Yaskawa INFORM job: Print3D.JBI

/JOB
//NAME Print3D
//POS
///NPOS 538,0,0,0,0,0
///TOOL 9
///POSTYPE PULSE
///PULSE
C00000=-32438,37072,-110539,-86183,-121616,78041,0
C00001=-32438,56188,-108455,-81750,-115935,87656,0
C00002=-32438,56821,-108216,-81665,-115782,87885,0
C00003=-32406,57586,-105976,-81950,-116211,87210,0
C00004=-32348,57787,-105393,-82074,-116292,87030,0
C00005=-31898,58636,-102954,-82798,-116500,86260,0
C00006=-31753,58820,-102432,-83000,-116512,86091,0
C00007=-30966,59540,-100399,-83997,-116406,85414,0
C00008=-30755,59682,-100001,-84246,-116346,85275,0
C00009=-29730,60178,-98619,-85379,-115942,84773,0
C00010=-29476,60259,-98393,-85644,-115819,84683,0
C00011=-28322,60462,-97831,-86792,-115175,84417,0
C00012=-28051,60472,-97803,-87049,-115007,84386,0
C00013=-26882,60354,-98131,-88113,-114216,84389,0
C00014=-26621,60290,-98306,-88341,-114026,84422,0
C00015=-25550,59868,-99482,-89239,-113195,84693,0
C00016=-25325,59740,-99839,-89419,-113009,84784,0
C00017=-24465,59071,-101720,-90078,-112243,85290,0
C00018=-24300,58897,-102214,-90195,-112083,85429,0
C00019=-20558,65330,-84764,-76831,-126138,82193,0
C00020=-20473,65073,-85436,-76785,-125928,82368,0
C00021=-20281,63933,-88440,-76413,-125114,83185,0
C00022=-20280,63674,-89129,-76290,-124955,83380,0
C00023=-20473,62589,-92031,-75590,-124397,84229,0
C00024=-20562,62357,-92656,-75394,-124304,84420,0
C00025=-20633,62241,-92968,-75270,-124274,84519,0
C00026=-21140,61448,-95121,-74399,-124058,85205,0
C00027=-21314,61269,-95612,-74142,-124041,85371,0
C00028=-22223,60633,-97359,-72935,-124133,86005,0
C00029=-22461,60524,-97659,-72644,-124194,86127,0
C00030=-23585,60225,-98488,-71363,-124621,86540,0
C00031=-23855,60198,-98563,-71076,-124755,86605,0
C00032=-25034,60265,-98378,-69905,-125482,86749,0
C00033=-25297,60322,-98219,-69665,-125679,86750,0
C00034=-30759,54831,-114236,-82744,-113724,89580,0
C00035=-30996,54948,-113875,-82536,-113911,89487,0
C00036=-31840,55566,-111976,-81865,-114711,88973,0
C00037=-31986,55730,-111478,-81769,-114886,88834,0
C00038=-32400,56520,-109107,-81604,-115582,88151,0
C00039=-32443,56714,-108532,-81625,-115721,87982,0
C00040=-32441,56759,-108398,-81642,-115746,87941,0
C00041=-26549,59218,-101304,-88131,-113571,85310,0
C00042=-26104,59051,-101778,-88513,-113235,85419,0
C00043=-25336,58461,-103455,-89105,-112549,85871,0
C00044=-24860,57729,-105559,-89395,-111996,86479,0
C00045=-21345,63810,-88769,-75336,-125745,83446,0
C00046=-21533,62838,-91363,-74678,-125240,84207,0
C00047=-22059,62019,-93570,-73765,-125019,84912,0
C00048=-22866,61443,-95135,-72683,-125107,85482,0
C00049=-23853,61172,-95878,-71559,-125500,85853,0
C00050=-24885,61232,-95712,-70546,-126159,85983,0
C00051=-30057,55478,-112245,-83650,-113759,88907,0
C00052=-30815,56036,-110556,-83049,-114467,88450,0
C00053=-31204,56744,-108442,-82877,-115075,87841,0
C00054=-31195,57522,-106160,-83130,-115500,87151,0
C00055=-30810,58276,-103983,-83747,-115680,86464,0
C00056=-30111,58912,-102170,-84625,-115587,85860,0
C00057=-29186,59348,-100939,-85647,-115233,85412,0
C00058=-28137,59526,-100438,-86701,-114669,85174,0
C00059=-27073,59422,-100730,-87686,-113973,85177,0
C00060=-26627,59248,-101220,-88065,-113630,85290,0
C00061=-26503,59292,-101097,-88193,-113572,85244,0
C00062=-26043,59118,-101588,-88588,-113223,85358,0
C00063=-25248,58507,-103322,-89200,-112515,85825,0
C00064=-24755,57750,-105498,-89502,-111944,86454,0
C00065=-21248,63808,-88772,-75428,-125681,83432,0
C00066=-21442,62804,-91454,-74751,-125159,84218,0
C00067=-21984,61958,-93735,-73809,-124930,84946,0
C00068=-22819,61364,-95353,-72691,-125021,85536,0
C00069=-23841,61083,-96120,-71527,-125427,85919,0
C00070=-24910,61146,-95949,-70477,-126107,86053,0
C00071=-30130,55424,-112411,-83560,-113765,88964,0
C00072=-30914,56000,-110664,-82939,-114497,88492,0
C00073=-31314,56732,-108479,-82763,-115127,87862,0
C00074=-31302,57536,-106119,-83029,-115568,87149,0
C00075=-30903,58316,-103868,-83669,-115753,86438,0
C00076=-30180,58974,-101994,-84577,-115657,85813,0
C00077=-29224,59426,-100721,-85633,-115291,85350,0
C00078=-28141,59610,-100203,-86721,-114708,85105,0
C00079=-27043,59502,-100505,-87735,-113986,85108,0
C00080=-26582,59322,-101013,-88127,-113631,85225,0
C00081=-26458,59365,-100890,-88255,-113573,85179,0
C00082=-25982,59185,-101398,-88663,-113212,85297,0
C00083=-25161,58554,-103189,-89294,-112480,85779,0
C00084=-21320,64890,-85917,-75895,-126401,82640,0
C00085=-21152,63807,-88776,-75520,-125616,83417,0
C00086=-21351,62770,-91544,-74823,-125078,84229,0
C00087=-21910,61897,-93900,-73853,-124843,84981,0
C00088=-22772,61284,-95570,-72699,-124936,85589,0
C00089=-23829,60995,-96362,-71495,-125353,85984,0
C00090=-24935,61060,-96185,-70408,-126055,86123,0
C00091=-30204,55370,-112576,-83469,-113771,89021,0
C00092=-31012,55964,-110771,-82828,-114527,88533,0
C00093=-31424,56720,-108515,-82649,-115180,87883,0
C00094=-31410,57551,-106078,-82927,-115635,87146,0
C00095=-30995,58356,-103753,-83591,-115828,86412,0
C00096=-30249,59037,-101817,-84530,-115728,85767,0
C00097=-29263,59503,-100502,-85620,-115350,85289,0
C00098=-28146,59694,-99968,-86740,-114746,85036,0
C00099=-27014,59583,-100279,-87785,-114000,85038,0
C00100=-26536,59395,-100806,-88189,-113632,85159,0
C00101=-26414,59439,-100683,-88316,-113573,85114,0
C00102=-25921,59252,-101208,-88737,-113200,85235,0
C00103=-25074,58601,-103056,-89388,-112445,85733,0
C00104=-21231,64924,-85829,-75997,-126360,82601,0
C00105=-21056,63806,-88778,-75612,-125552,83403,0
C00106=-21259,62736,-91634,-74896,-124997,84240,0
C00107=-21835,61837,-94064,-73898,-124755,85015,0
C00108=-22725,61205,-95786,-72707,-124850,85642,0
C00109=-23817,60907,-96603,-71464,-125280,86050,0
C00110=-24961,60974,-96420,-70339,-126003,86193,0
C00111=-30277,55316,-112741,-83379,-113776,89078,0
C00112=-31111,55928,-110879,-82718,-114558,88574,0
C00113=-31534,56708,-108550,-82535,-115232,87903,0
C00114=-31517,57565,-106036,-82825,-115703,87144,0
C00115=-31088,58397,-103638,-83513,-115903,86386,0
C00116=-30317,59099,-101640,-84484,-115799,85720,0
C00117=-29301,59581,-100284,-85607,-115409,85227,0
C00118=-28150,59778,-99732,-86759,-114784,84966,0
C00119=-26984,59663,-100054,-87834,-114014,84969,0
C00120=-26491,59469,-100598,-88250,-113633,85094,0
C00121=-26332,59013,-101884,-88286,-113359,85467,0
C00122=-24985,57748,-105506,-89278,-112076,86471,0
C00123=-24944,57669,-105734,-89300,-112022,86537,0
C00124=-21511,64356,-87324,-75447,-126200,83067,0
C00125=-25467,58473,-103419,-88982,-112632,85869,0
C00126=-25645,58607,-103036,-88843,-112789,85766,0
C00127=-21453,63977,-88326,-75315,-125923,83339,0
C00128=-21420,63763,-88894,-75241,-125765,83493,0
C00129=-21433,63691,-89084,-75193,-125729,83550,0
C00130=-25822,58743,-102651,-88706,-112947,85662,0
C00131=-25998,58879,-102263,-88572,-113105,85557,0
C00132=-21465,63524,-89527,-75080,-125643,83679,0
C00133=-21497,63359,-89968,-74968,-125557,83808,0
C00134=-26173,59017,-101873,-88439,-113264,85453,0
C00135=-26184,59026,-101848,-88430,-113274,85446,0
C00136=-26310,59073,-101715,-88322,-113368,85415,0
C00137=-21529,63194,-90407,-74856,-125472,83937,0
C00138=-21562,63031,-90844,-74745,-125386,84066,0
C00139=-26443,59123,-101573,-88207,-113470,85382,0
C00140=-26577,59174,-101429,-88093,-113571,85349,0
C00141=-21595,62868,-91280,-74634,-125299,84193,0
C00142=-21603,62825,-91397,-74604,-125276,84227,0
C00143=-21648,62753,-91590,-74525,-125258,84289,0
C00144=-26710,59225,-101285,-87979,-113672,85316,0
C00145=-26843,59277,-101140,-87866,-113774,85282,0
C00146=-21710,62654,-91854,-74417,-125232,84374,0
C00147=-21772,62557,-92118,-74308,-125205,84457,0
C00148=-26976,59328,-100994,-87753,-113876,85249,0
C00149=-27108,59381,-100847,-87641,-113978,85215,0
C00150=-21835,62459,-92380,-74200,-125179,84541,0
C00151=-21897,62362,-92642,-74091,-125153,84625,0
C00152=-27224,59395,-100808,-87534,-114055,85212,0
C00153=-27339,59405,-100778,-87428,-114129,85212,0
C00154=-21960,62265,-92903,-73983,-125127,84708,0
C00155=-22023,62169,-93163,-73874,-125101,84791,0
C00156=-27453,59416,-100747,-87322,-114204,85212,0
C00157=-27568,59427,-100716,-87216,-114278,85212,0
C00158=-22086,62073,-93422,-73765,-125074,84875,0
C00159=-22112,62034,-93528,-73720,-125063,84909,0
C00160=-22159,61999,-93623,-73656,-125068,84943,0
C00161=-27682,59438,-100685,-87110,-114353,85212,0
C00162=-27796,59450,-100653,-87005,-114428,85211,0
C00163=-22240,61941,-93782,-73548,-125078,85001,0
C00164=-22321,61882,-93941,-73440,-125087,85058,0
C00165=-27910,59461,-100621,-86899,-114503,85210,0
C00166=-28024,59473,-100588,-86794,-114578,85210,0
C00167=-22402,61824,-94100,-73331,-125095,85116,0
C00168=-22483,61766,-94257,-73222,-125104,85173,0
C00169=-28138,59485,-100555,-86688,-114653,85209,0
C00170=-28149,59486,-100552,-86678,-114660,85209,0
C00171=-28242,59469,-100598,-86585,-114710,85231,0
C00172=-22564,61708,-94415,-73113,-125113,85231,0
C00173=-22645,61650,-94572,-73004,-125122,85288,0
C00174=-28344,59452,-100648,-86483,-114765,85254,0
C00175=-28446,59434,-100698,-86380,-114820,85277,0
C00176=-22727,61592,-94728,-72895,-125130,85346,0
C00177=-22809,61535,-94884,-72785,-125140,85402,0
C00178=-28549,59416,-100747,-86277,-114875,85300,0
C00179=-28651,59399,-100796,-86174,-114929,85324,0
C00180=-22891,61478,-95039,-72675,-125149,85459,0
C00181=-22987,61451,-95114,-72566,-125187,85496,0
C00182=-28754,59382,-100845,-86071,-114985,85347,0
C00183=-28856,59364,-100893,-85968,-115040,85370,0
C00184=-23082,61424,-95188,-72457,-125225,85532,0
C00185=-23179,61397,-95262,-72348,-125263,85569,0
C00186=-28959,59347,-100941,-85865,-115095,85393,0
C00187=-29062,59331,-100988,-85761,-115150,85416,0
C00188=-23275,61370,-95335,-72238,-125302,85606,0
C00189=-23371,61343,-95408,-72129,-125340,85642,0
C00190=-29164,59314,-101036,-85658,-115204,85438,0
C00191=-29257,59269,-101162,-85556,-115240,85484,0
C00192=-23467,61317,-95480,-72019,-125379,85678,0
C00193=-23564,61291,-95552,-71909,-125417,85714,0
C00194=-29349,59224,-101287,-85454,-115276,85530,0
C00195=-29442,59180,-101412,-85351,-115312,85575,0
C00196=-23660,61264,-95623,-71799,-125454,85750,0
C00197=-23757,61239,-95694,-71689,-125494,85786,0
C00198=-29535,59136,-101537,-85249,-115348,85620,0
C00199=-29628,59092,-101661,-85146,-115383,85665,0
C00200=-23855,61216,-95757,-71579,-125535,85820,0
C00201=-23966,61222,-95741,-71470,-125605,85834,0
C00202=-29721,59048,-101784,-85043,-115418,85710,0
C00203=-29815,59005,-101908,-84939,-115453,85755,0
C00204=-24076,61228,-95725,-71362,-125675,85848,0
C00205=-24187,61234,-95708,-71253,-125746,85862,0
C00206=-29908,58961,-102031,-84836,-115489,85800,0
C00207=-30002,58918,-102153,-84732,-115525,85845,0
C00208=-24298,61240,-95691,-71144,-125816,85876,0
C00209=-24409,61246,-95673,-71036,-125888,85890,0
C00210=-30091,58861,-102314,-84628,-115550,85901,0
C00211=-30173,58785,-102531,-84525,-115561,85973,0
C00212=-24519,61253,-95655,-70927,-125959,85904,0
C00213=-24630,61260,-95636,-70819,-126029,85918,0
C00214=-30256,58709,-102748,-84422,-115573,86045,0
C00215=-30338,58633,-102964,-84318,-115584,86117,0
C00216=-24741,61267,-95617,-70711,-126100,85931,0
C00217=-24841,61273,-95599,-70612,-126165,85944,0
C00218=-24853,61278,-95586,-70603,-126176,85942,0
C00219=-30421,58557,-103180,-84214,-115595,86188,0
C00220=-30504,58482,-103395,-84110,-115606,86260,0
C00221=-24982,61330,-95443,-70498,-126292,85925,0
C00222=-29264,55260,-112912,-84393,-113237,89051,0
C00223=-30587,58407,-103609,-84006,-115617,86331,0
C00224=-30671,58332,-103822,-83900,-115628,86403,0
C00225=-29407,55307,-112767,-84261,-113335,89018,0
C00226=-29550,55355,-112622,-84129,-113433,88983,0
C00227=-30749,58243,-104079,-83796,-115628,86487,0
C00228=-30814,58113,-104451,-83692,-115598,86604,0
C00229=-29693,55402,-112476,-83998,-113532,88949,0
C00230=-29835,55450,-112329,-83868,-113631,88915,0
C00231=-30878,57985,-104821,-83589,-115567,86721,0
C00232=-30943,57857,-105191,-83485,-115537,86837,0
C00233=-29979,55504,-112166,-83737,-113734,88876,0
C00234=-30155,55630,-111781,-83595,-113896,88772,0
C00235=-31008,57729,-105559,-83380,-115507,86954,0
C00236=-31074,57603,-105926,-83275,-115476,87070,0
C00237=-30331,55758,-111394,-83455,-114058,88667,0
C00238=-30505,55887,-111005,-83317,-114221,88561,0
C00239=-31104,57379,-106577,-83175,-115372,87269,0
C00240=-31107,57086,-107436,-83081,-115213,87528,0
C00241=-30678,56016,-110613,-83182,-114384,88456,0
C00242=-30701,56034,-110561,-83164,-114406,88443,0
C00243=-31079,56718,-108521,-82994,-114993,87854,0
C00244=-31110,56796,-108290,-82988,-115053,87786,0
C00245=-31110,56739,-108311,-82995,-115066,87766,0
C00246=-27205,58149,-104211,-87244,-113559,86206,0
C00247=-26990,58071,-104437,-87431,-113400,86258,0
C00248=-26590,57768,-105309,-87742,-113042,86493,0
C00249=-26353,57390,-106405,-87879,-112748,86810,0
C00250=-26309,56984,-107592,-87822,-112552,87169,0
C00251=-26470,56599,-108727,-87568,-112474,87528,0
C00252=-23096,62855,-91200,-73195,-126301,84395,0
C00253=-23513,62550,-92020,-72630,-126351,84695,0
C00254=-27912,55978,-110579,-85973,-112960,88201,0
C00255=-28512,56029,-110426,-85386,-113301,88198,0
C00256=-29044,56212,-109879,-84904,-113676,88071,0
C00257=-29441,56506,-109003,-84591,-114041,87834,0
C00258=-29655,56877,-107905,-84486,-114350,87518,0
C00259=-29666,57283,-106718,-84594,-114563,87159,0
C00260=-29477,57673,-105584,-84894,-114651,86801,0
C00261=-29117,58000,-104641,-85342,-114603,86487,0
C00262=-28629,58223,-104001,-85882,-114424,86254,0
C00263=-28070,58314,-103740,-86449,-114138,86131,0
C00264=-27502,58261,-103892,-86985,-113781,86132,0
C00265=-27284,58179,-104126,-87174,-113618,86186,0
C00266=-26842,58698,-102644,-87736,-113572,85707,0
C00267=-26501,58571,-103006,-88032,-113317,85791,0
C00268=-25900,58112,-104318,-88496,-112779,86144,0
C00269=-25534,57541,-105965,-88714,-112342,86620,0
C00270=-21963,63771,-88757,-74759,-126177,83521,0
C00271=-22119,63009,-90789,-74229,-125779,84117,0
C00272=-22533,62364,-92520,-73503,-125606,84671,0
C00273=-23163,61909,-93748,-72655,-125679,85119,0
C00274=-23928,61694,-94331,-71784,-125991,85410,0
C00275=-28785,55501,-112019,-84967,-113169,88710,0
C00276=-29592,55774,-111193,-84229,-113731,88518,0
C00277=-30187,56213,-109873,-83759,-114282,88162,0
C00278=-30500,56770,-108221,-83613,-114753,87685,0
C00279=-30503,57380,-106435,-83795,-115080,87146,0
C00280=-30210,57968,-104731,-84264,-115217,86608,0
C00281=-29665,58463,-103313,-84945,-115144,86135,0
C00282=-28937,58802,-102350,-85750,-114870,85785,0
C00283=-28107,58940,-101958,-86587,-114434,85600,0
C00284=-27265,58860,-102186,-87373,-113892,85602,0
C00285=-26921,58728,-102560,-87668,-113632,85688,0
C00286=-26527,59199,-101227,-88167,-113580,85259,0
C00287=-26075,59029,-101709,-88555,-113238,85371,0
C00288=-25294,58428,-103413,-89156,-112541,85830,0
C00289=-24810,57684,-105551,-89451,-111980,86446,0
C00290=-21298,63758,-88793,-75392,-125729,83423,0
C00291=-21490,62770,-91428,-74724,-125217,84195,0
C00292=-22023,61938,-93671,-73797,-124993,84911,0
C00293=-22843,61353,-95261,-72698,-125083,85490,0
C00294=-23847,61077,-96016,-71555,-125482,85867,0
C00295=-24897,61138,-95847,-70525,-126152,85999,0
C00296=-30092,55394,-112346,-83613,-113775,88913,0
C00297=-30862,55961,-110629,-83003,-114494,88449,0
C00298=-31257,56682,-108482,-82829,-115113,87830,0
C00299=-31246,57473,-106163,-83089,-115545,87131,0
C00300=-30855,58241,-103950,-83717,-115727,86432,0
C00301=-30144,58888,-102107,-84609,-115631,85818,0
C00302=-29204,59331,-100856,-85647,-115272,85363,0
C00303=-28139,59513,-100347,-86717,-114697,85122,0
C00304=-27058,59407,-100644,-87716,-113988,85125,0
C00305=-26605,59229,-101142,-88100,-113640,85239,0
C00306=-26453,58811,-102323,-88139,-113383,85582,0
C00307=-26840,57508,-106061,-87432,-113075,86739,0
C00308=-29262,56973,-107624,-84903,-114183,87400,0
C00309=-28112,56493,-109040,-85911,-113318,87742,0
C00310=-27221,56686,-108470,-86846,-112924,87502,0
C00311=-27221,56629,-108492,-86852,-112935,87482,0
C00312=-27205,58094,-104232,-87250,-113569,86186,0
C00313=-26990,58016,-104458,-87437,-113410,86238,0
C00314=-26590,57712,-105331,-87747,-113051,86473,0
C00315=-26353,57334,-106427,-87885,-112757,86789,0
C00316=-26309,56928,-107613,-87827,-112561,87149,0
C00317=-26470,56542,-108748,-87574,-112484,87508,0
C00318=-23096,62804,-91222,-73207,-126316,84377,0
C00319=-23513,62498,-92041,-72641,-126367,84677,0
C00320=-27912,55921,-110600,-85979,-112971,88180,0
C00321=-28512,55972,-110448,-85392,-113313,88177,0
C00322=-29044,56155,-109900,-84910,-113688,88050,0
C00323=-29441,56449,-109024,-84598,-114053,87814,0
C00324=-29655,56821,-107926,-84492,-114362,87497,0
C00325=-29666,57227,-106739,-84601,-114574,87139,0
C00326=-29477,57617,-105606,-84901,-114663,86781,0
C00327=-29117,57944,-104663,-85349,-114614,86467,0
C00328=-28629,58168,-104022,-85888,-114435,86235,0
C00329=-28070,58259,-103762,-86456,-114148,86111,0
C00330=-27502,58206,-103914,-86991,-113791,86113,0
C00331=-27284,58124,-104148,-87180,-113628,86167,0
C00332=-26842,58644,-102666,-87742,-113582,85687,0
C00333=-26501,58517,-103027,-88037,-113326,85771,0
C00334=-25900,58057,-104339,-88502,-112788,86124,0
C00335=-25534,57486,-105986,-88720,-112351,86600,0
C00336=-21963,63721,-88780,-74770,-126192,83504,0
C00337=-22119,62957,-90811,-74240,-125795,84099,0
C00338=-22533,62312,-92541,-73514,-125622,84653,0
C00339=-23163,61857,-93769,-72666,-125695,85101,0
C00340=-23928,61642,-94352,-71796,-126007,85393,0
C00341=-28785,55444,-112040,-84973,-113181,88689,0
C00342=-29592,55716,-111215,-84235,-113743,88497,0
C00343=-30187,56156,-109895,-83765,-114295,88141,0
C00344=-30500,56714,-108242,-83620,-114765,87665,0
C00345=-30503,57324,-106457,-83802,-115093,87126,0
C00346=-30210,57913,-104753,-84271,-115228,86588,0
C00347=-29665,58409,-103334,-84952,-115155,86116,0
C00348=-28937,58748,-102371,-85756,-114881,85766,0
C00349=-28107,58886,-101980,-86594,-114444,85580,0
C00350=-27265,58805,-102208,-87379,-113902,85582,0
C00351=-26921,58674,-102581,-87674,-113641,85668,0
C00352=-26527,59146,-101248,-88173,-113589,85239,0
C00353=-26075,58975,-101730,-88560,-113247,85351,0
C00354=-25294,58374,-103434,-89162,-112550,85809,0
C00355=-24810,57629,-105573,-89457,-111988,86427,0
C00356=-21298,63707,-88815,-75403,-125743,83405,0
C00357=-21490,62718,-91450,-74735,-125232,84178,0
C00358=-22023,61886,-93693,-73808,-125009,84894,0
C00359=-22843,61300,-95283,-72709,-125099,85473,0
C00360=-23847,61024,-96037,-71567,-125499,85849,0
C00361=-24897,61086,-95869,-70537,-126170,85982,0
C00362=-30092,55336,-112368,-83620,-113787,88892,0
C00363=-30862,55904,-110651,-83010,-114507,88429,0
C00364=-31257,56625,-108503,-82837,-115126,87810,0
C00365=-31246,57418,-106184,-83096,-115558,87110,0
C00366=-30855,58186,-103971,-83724,-115738,86412,0
C00367=-30144,58834,-102129,-84616,-115643,85799,0
C00368=-29204,59277,-100877,-85654,-115282,85344,0
C00369=-28139,59459,-100369,-86723,-114707,85103,0
C00370=-27058,59353,-100665,-87722,-113997,85105,0
C00371=-26605,59176,-101164,-88106,-113649,85220,0
C00372=-26453,58757,-102345,-88144,-113392,85563,0
C00373=-27718,56871,-107781,-86424,-113319,87301,0
C00374=-27564,56939,-107579,-86595,-113265,87227,0
C00375=-27389,57100,-107108,-86810,-113240,87071,0
C00376=-27305,57295,-106542,-86942,-113280,86893,0
C00377=-27322,57499,-105949,-86979,-113380,86714,0
C00378=-27436,57688,-105402,-86918,-113528,86557,0
C00379=-27631,57840,-104965,-86768,-113707,86439,0
C00380=-27886,57935,-104691,-86546,-113897,86376,0
C00381=-28169,57961,-104614,-86278,-114073,86376,0
C00382=-28207,57955,-104632,-86239,-114092,86384,0
C00383=-27428,56276,-109538,-86556,-112883,87818,0
C00384=-27520,56237,-109655,-86454,-112914,87860,0
C00385=-27810,56193,-109785,-86153,-113049,87921,0
C00386=-28106,56218,-109712,-85865,-113219,87920,0
C00387=-28369,56308,-109444,-85627,-113405,87858,0
C00388=-28569,56453,-109014,-85468,-113584,87742,0
C00389=-28656,56596,-108590,-85421,-113702,87619,0
C00390=-28925,57203,-106808,-85324,-114149,87099,0
C00391=-28925,57147,-106829,-85331,-114160,87078,0
C00392=-27205,58040,-104254,-87256,-113579,86166,0
C00393=-26990,57961,-104480,-87443,-113420,86218,0
C00394=-26590,57657,-105352,-87753,-113061,86453,0
C00395=-26353,57279,-106448,-87890,-112767,86769,0
C00396=-26309,56872,-107635,-87833,-112571,87128,0
C00397=-26470,56486,-108770,-87579,-112494,87487,0
C00398=-23096,62752,-91244,-73218,-126332,84360,0
C00399=-23513,62447,-92063,-72653,-126384,84660,0
C00400=-27912,55863,-110622,-85985,-112982,88159,0
C00401=-28512,55914,-110469,-85398,-113324,88156,0
C00402=-29044,56098,-109922,-84917,-113700,88029,0
C00403=-29441,56392,-109046,-84604,-114065,87793,0
C00404=-29655,56765,-107948,-84499,-114373,87477,0
C00405=-29666,57171,-106761,-84607,-114586,87118,0
C00406=-29477,57562,-105627,-84908,-114674,86761,0
C00407=-29117,57889,-104684,-85356,-114625,86447,0
C00408=-28629,58113,-104044,-85895,-114445,86215,0
C00409=-28070,58204,-103784,-86462,-114158,86091,0
C00410=-27502,58151,-103935,-86997,-113801,86093,0
C00411=-27284,58069,-104169,-87187,-113638,86146,0
C00412=-26842,58589,-102687,-87748,-113591,85668,0
C00413=-26501,58462,-103049,-88043,-113335,85751,0
C00414=-25900,58002,-104361,-88508,-112797,86104,0
C00415=-25534,57430,-106008,-88725,-112360,86579,0
C00416=-21963,63670,-88802,-74782,-126207,83487,0
C00417=-22119,62906,-90833,-74252,-125810,84082,0
C00418=-22533,62261,-92563,-73526,-125637,84636,0
C00419=-23163,61805,-93791,-72678,-125711,85084,0
C00420=-23928,61590,-94374,-71807,-126024,85375,0
C00421=-28785,55386,-112062,-84979,-113193,88668,0
C00422=-29592,55659,-111236,-84242,-113756,88476,0
C00423=-30187,56099,-109917,-83772,-114307,88120,0
C00424=-30500,56657,-108264,-83627,-114778,87645,0
C00425=-30503,57268,-106478,-83809,-115104,87106,0
C00426=-30210,57858,-104774,-84278,-115240,86568,0
C00427=-29665,58354,-103356,-84959,-115166,86096,0
C00428=-28937,58693,-102393,-85763,-114891,85746,0
C00429=-28107,58832,-102001,-86600,-114454,85561,0
C00430=-27265,58751,-102229,-87385,-113911,85563,0
C00431=-26921,58619,-102603,-87680,-113650,85649,0
C00432=-26527,59092,-101270,-88179,-113598,85220,0
C00433=-26075,58920,-101752,-88566,-113256,85331,0
C00434=-25294,58319,-103456,-89167,-112558,85790,0
C00435=-24810,57573,-105595,-89462,-111997,86406,0
C00436=-21298,63656,-88837,-75414,-125758,83388,0
C00437=-21490,62667,-91472,-74746,-125246,84160,0
C00438=-22023,61834,-93715,-73819,-125025,84876,0
C00439=-22843,61248,-95305,-72721,-125117,85455,0
C00440=-23847,60972,-96059,-71578,-125517,85832,0
C00441=-24897,61033,-95890,-70548,-126188,85964,0
C00442=-30092,55278,-112390,-83626,-113800,88871,0
C00443=-30862,55847,-110672,-83017,-114520,88408,0
C00444=-31257,56569,-108525,-82844,-115138,87790,0
C00445=-31246,57362,-106206,-83103,-115569,87090,0
C00446=-30855,58131,-103993,-83731,-115751,86392,0
C00447=-30144,58779,-102150,-84623,-115653,85779,0
C00448=-29204,59224,-100899,-85661,-115292,85325,0
C00449=-28139,59405,-100391,-86730,-114717,85084,0
C00450=-27058,59299,-100687,-87728,-114007,85086,0
C00451=-26605,59122,-101185,-88112,-113658,85201,0
C00452=-26453,58703,-102366,-88150,-113401,85543,0
C00453=-26840,57397,-106104,-87444,-113094,86699,0
C00454=-29262,56861,-107667,-84916,-114206,87360,0
C00455=-28112,56380,-109083,-85924,-113341,87701,0
C00456=-27221,56573,-108513,-86858,-112945,87461,0
C00457=-27221,56516,-108535,-86864,-112956,87440,0
C00458=-27205,57985,-104275,-87262,-113588,86146,0
C00459=-26990,57906,-104501,-87449,-113429,86198,0
C00460=-26590,57602,-105374,-87759,-113070,86433,0
C00461=-26353,57223,-106469,-87896,-112776,86749,0
C00462=-26309,56816,-107656,-87839,-112581,87107,0
C00463=-26470,56429,-108792,-87585,-112504,87466,0
C00464=-23096,62701,-91265,-73230,-126349,84343,0
C00465=-23513,62395,-92085,-72665,-126400,84643,0
C00466=-27912,55806,-110644,-85991,-112993,88137,0
C00467=-28512,55857,-110491,-85405,-113336,88136,0
C00468=-29044,56041,-109943,-84923,-113711,88008,0
C00469=-29441,56336,-109067,-84611,-114076,87773,0
C00470=-29655,56709,-107969,-84506,-114385,87457,0
C00471=-29666,57115,-106782,-84614,-114598,87099,0
C00472=-29477,57507,-105649,-84914,-114685,86741,0
C00473=-29117,57834,-104705,-85362,-114636,86427,0
C00474=-28629,58058,-104065,-85901,-114456,86195,0
C00475=-28070,58149,-103805,-86468,-114168,86072,0
C00476=-27502,58096,-103957,-87003,-113811,86073,0
C00477=-27284,58014,-104191,-87193,-113648,86127,0
C00478=-26842,58535,-102709,-87754,-113600,85648,0
C00479=-26501,58408,-103070,-88049,-113344,85731,0
C00480=-25900,57947,-104382,-88513,-112806,86084,0
C00481=-25534,57375,-106029,-88730,-112369,86559,0
C00482=-21963,63619,-88824,-74793,-126222,83470,0
C00483=-22119,62855,-90854,-74263,-125824,84065,0
C00484=-22533,62209,-92585,-73537,-125653,84619,0
C00485=-23163,61754,-93813,-72689,-125728,85067,0
C00486=-23928,61538,-94396,-71819,-126042,85358,0
C00487=-28785,55328,-112084,-84986,-113205,88647,0
C00488=-29592,55601,-111258,-84248,-113768,88455,0
C00489=-30187,56042,-109938,-83779,-114320,88100,0
C00490=-30500,56601,-108285,-83634,-114790,87624,0
C00491=-30503,57212,-106500,-83816,-115117,87085,0
C00492=-30210,57803,-104796,-84285,-115251,86548,0
C00493=-29665,58300,-103377,-84965,-115178,86076,0
C00494=-28937,58639,-102414,-85770,-114902,85726,0
C00495=-28107,58778,-102023,-86607,-114464,85541,0
C00496=-27265,58697,-102251,-87392,-113921,85543,0
C00497=-26921,58565,-102624,-87686,-113660,85629,0
C00498=-26527,59038,-101291,-88185,-113607,85201,0
C00499=-26075,58866,-101773,-88572,-113264,85312,0
C00500=-25294,58264,-103477,-89172,-112567,85770,0
C00501=-24810,57518,-105616,-89467,-112005,86386,0
C00502=-21298,63606,-88859,-75425,-125773,83371,0
C00503=-21490,62616,-91494,-74758,-125261,84143,0
C00504=-22023,61782,-93736,-73831,-125041,84858,0
C00505=-22843,61196,-95326,-72732,-125133,85437,0
C00506=-23847,60919,-96081,-71590,-125534,85814,0
C00507=-24897,60981,-95912,-70560,-126206,85946,0
C00508=-30092,55220,-112411,-83633,-113813,88849,0
C00509=-30862,55789,-110694,-83024,-114533,88387,0
C00510=-31257,56513,-108546,-82851,-115151,87769,0
C00511=-31246,57307,-106227,-83110,-115582,87070,0
C00512=-30855,58076,-104014,-83738,-115762,86373,0
C00513=-30144,58725,-102171,-84630,-115665,85760,0
C00514=-29204,59170,-100920,-85668,-115303,85305,0
C00515=-28139,59351,-100412,-86736,-114727,85064,0
C00516=-27058,59245,-100708,-87734,-114016,85067,0
C00517=-26605,59068,-101207,-88118,-113667,85181,0
C00518=-26453,58648,-102388,-88156,-113411,85523,0
C00519=-27723,56756,-107830,-86431,-113342,87262,0
C00520=-27564,56827,-107622,-86607,-113286,87187,0
C00521=-27389,56989,-107151,-86821,-113261,87030,0
C00522=-27305,57183,-106585,-86954,-113300,86852,0
C00523=-27322,57388,-105992,-86991,-113400,86674,0
C00524=-27436,57577,-105445,-86930,-113548,86517,0
C00525=-27631,57729,-105008,-86780,-113728,86399,0
C00526=-27886,57824,-104734,-86558,-113917,86337,0
C00527=-28169,57851,-104657,-86290,-114094,86336,0
C00528=-28212,57844,-104677,-86246,-114116,86345,0
C00529=-27432,56160,-109587,-86563,-112906,87778,0
C00530=-27520,56123,-109699,-86466,-112936,87818,0
C00531=-27810,56079,-109828,-86165,-113071,87880,0
C00532=-28106,56104,-109755,-85877,-113242,87878,0
C00533=-28369,56194,-109487,-85639,-113428,87816,0
C00534=-28569,56340,-109057,-85481,-113607,87700,0
C00535=-28679,56522,-108517,-85421,-113757,87544,0
C00536=-28948,57132,-106733,-85326,-114204,87024,0
C00537=-28948,38167,-109035,-89068,-118868,77542,0
//INST
///DATE 2024/05/09 11:40
///COMM Generated using RoboDK
///ATTR SC,RW
///GROUP1 RB1
NOP
'Program generated by RoboDK v
'5.5.3 for Yaskawa SIA10D on 0
'9/05/2024 11:40:04
'Using nominal kinematics.
'MCodeHandler(107)
'MCodeHandler(104)
'Using Printing Frame (targets
' wrt base):
'467.9,0.0,-338.7,0.0,0.0,180.
'0
'Tool MDPH2 should be close to
':
'-231.5,0.0,70.1,0.0,-90.0,0.0
'Show MDPH2
MOVJ C00000 VJ=50.00 PL=1
MOVL C00001 V=83.3 PL=1
'MCodeHandler(109)
'MCodeHandler(82)
'ExtruderHandler(0.00000)
MOVL C00002 V=130.0 PL=1
'ExtruderHandler(-2.00000)
'ExtruderHandler(0.00000)
'ExtruderHandler(2.00000)
'ExtruderHandler(2.14392)
MOVL C00003 V=30.0 PL=1
'ExtruderHandler(2.18171)
MOVL C00004 V=30.0 PL=1
'ExtruderHandler(2.34618)
MOVL C00005 V=30.0 PL=1
'ExtruderHandler(2.38397)
MOVL C00006 V=30.0 PL=1
'ExtruderHandler(2.54845)
MOVL C00007 V=30.0 PL=1
'ExtruderHandler(2.58624)
MOVL C00008 V=30.0 PL=1
'ExtruderHandler(2.75072)
MOVL C00009 V=30.0 PL=1
'ExtruderHandler(2.78851)
MOVL C00010 V=30.0 PL=1
'ExtruderHandler(2.95298)
MOVL C00011 V=30.0 PL=1
'ExtruderHandler(2.99077)
MOVL C00012 V=30.0 PL=1
'ExtruderHandler(3.15525)
MOVL C00013 V=30.0 PL=1
'ExtruderHandler(3.19304)
MOVL C00014 V=30.0 PL=1
'ExtruderHandler(3.35751)
MOVL C00015 V=30.0 PL=1
'ExtruderHandler(3.39530)
MOVL C00016 V=30.0 PL=1
'ExtruderHandler(3.55978)
MOVL C00017 V=30.0 PL=1
'ExtruderHandler(3.59757)
MOVL C00018 V=30.0 PL=1
'ExtruderHandler(3.76205)
MOVL C00019 V=30.0 PL=1
'ExtruderHandler(3.79984)
MOVL C00020 V=30.0 PL=1
'ExtruderHandler(3.96431)
MOVL C00021 V=30.0 PL=1
'ExtruderHandler(4.00210)
MOVL C00022 V=30.0 PL=1
'ExtruderHandler(4.16658)
MOVL C00023 V=30.0 PL=1
'ExtruderHandler(4.20437)
MOVL C00024 V=30.0 PL=1
'ExtruderHandler(4.22493)
MOVL C00025 V=30.0 PL=1
'ExtruderHandler(4.36885)
MOVL C00026 V=30.0 PL=1
'ExtruderHandler(4.40664)
MOVL C00027 V=30.0 PL=1
'ExtruderHandler(4.57111)
MOVL C00028 V=30.0 PL=1
'ExtruderHandler(4.60890)
MOVL C00029 V=30.0 PL=1
'ExtruderHandler(4.77338)
MOVL C00030 V=30.0 PL=1
'ExtruderHandler(4.81117)
MOVL C00031 V=30.0 PL=1
'ExtruderHandler(4.97564)
MOVL C00032 V=30.0 PL=1
'ExtruderHandler(5.01343)
MOVL C00033 V=30.0 PL=1
'ExtruderHandler(5.17791)
MOVL C00034 V=30.0 PL=1
'ExtruderHandler(5.21570)
MOVL C00035 V=30.0 PL=1
'ExtruderHandler(5.38018)
MOVL C00036 V=30.0 PL=1
'ExtruderHandler(5.41797)
MOVL C00037 V=30.0 PL=1
'ExtruderHandler(5.58244)
MOVL C00038 V=30.0 PL=1
'ExtruderHandler(5.62023)
MOVL C00039 V=30.0 PL=1
'ExtruderHandler(5.62895)
MOVL C00040 V=30.0 PL=1
'ExtruderHandler(3.62895)
'ExtruderHandler(0.00000)
MOVL C00041 V=130.0 PL=1
'ExtruderHandler(2.00000)
'ExtruderHandler(2.06711)
MOVL C00042 V=30.0 PL=1
'ExtruderHandler(2.21389)
MOVL C00043 V=30.0 PL=1
'ExtruderHandler(2.36067)
MOVL C00044 V=30.0 PL=1
'ExtruderHandler(2.50746)
MOVL C00045 V=30.0 PL=1
'ExtruderHandler(2.65424)
MOVL C00046 V=30.0 PL=1
'ExtruderHandler(2.80102)
MOVL C00047 V=30.0 PL=1
'ExtruderHandler(2.94781)
MOVL C00048 V=30.0 PL=1
'ExtruderHandler(3.09459)
MOVL C00049 V=30.0 PL=1
'ExtruderHandler(3.24138)
MOVL C00050 V=30.0 PL=1
'ExtruderHandler(3.38816)
MOVL C00051 V=30.0 PL=1
'ExtruderHandler(3.53494)
MOVL C00052 V=30.0 PL=1
'ExtruderHandler(3.68173)
MOVL C00053 V=30.0 PL=1
'ExtruderHandler(3.82851)
MOVL C00054 V=30.0 PL=1
'ExtruderHandler(3.97529)
MOVL C00055 V=30.0 PL=1
'ExtruderHandler(4.12208)
MOVL C00056 V=30.0 PL=1
'ExtruderHandler(4.26886)
MOVL C00057 V=30.0 PL=1
'ExtruderHandler(4.41565)
MOVL C00058 V=30.0 PL=1
'ExtruderHandler(4.56243)
MOVL C00059 V=30.0 PL=1
'ExtruderHandler(4.63027)
MOVL C00060 V=30.0 PL=1
MOVL C00061 V=130.0 PL=1
'ExtruderHandler(4.69986)
MOVL C00062 V=30.0 PL=1
'ExtruderHandler(4.85161)
MOVL C00063 V=30.0 PL=1
'ExtruderHandler(5.00336)
MOVL C00064 V=30.0 PL=1
'ExtruderHandler(5.15512)
MOVL C00065 V=30.0 PL=1
'ExtruderHandler(5.30687)
MOVL C00066 V=30.0 PL=1
'ExtruderHandler(5.45863)
MOVL C00067 V=30.0 PL=1
'ExtruderHandler(5.61038)
MOVL C00068 V=30.0 PL=1
'ExtruderHandler(5.76213)
MOVL C00069 V=30.0 PL=1
'ExtruderHandler(5.91389)
MOVL C00070 V=30.0 PL=1
'ExtruderHandler(6.06564)
MOVL C00071 V=30.0 PL=1
'ExtruderHandler(6.21739)
MOVL C00072 V=30.0 PL=1
'ExtruderHandler(6.36915)
MOVL C00073 V=30.0 PL=1
'ExtruderHandler(6.52090)
MOVL C00074 V=30.0 PL=1
'ExtruderHandler(6.67265)
MOVL C00075 V=30.0 PL=1
'ExtruderHandler(6.82441)
MOVL C00076 V=30.0 PL=1
'ExtruderHandler(6.97616)
MOVL C00077 V=30.0 PL=1
'ExtruderHandler(7.12791)
MOVL C00078 V=30.0 PL=1
'ExtruderHandler(7.27967)
MOVL C00079 V=30.0 PL=1
'ExtruderHandler(7.34999)
MOVL C00080 V=30.0 PL=1
MOVL C00081 V=130.0 PL=1
'ExtruderHandler(7.42207)
MOVL C00082 V=30.0 PL=1
'ExtruderHandler(7.57879)
MOVL C00083 V=30.0 PL=1
'ExtruderHandler(7.73551)
MOVL C00084 V=30.0 PL=1
'ExtruderHandler(7.89224)
MOVL C00085 V=30.0 PL=1
'ExtruderHandler(8.04896)
MOVL C00086 V=30.0 PL=1
'ExtruderHandler(8.20568)
MOVL C00087 V=30.0 PL=1
'ExtruderHandler(8.36241)
MOVL C00088 V=30.0 PL=1
'ExtruderHandler(8.51913)
MOVL C00089 V=30.0 PL=1
'ExtruderHandler(8.67585)
MOVL C00090 V=30.0 PL=1
'ExtruderHandler(8.83258)
MOVL C00091 V=30.0 PL=1
'ExtruderHandler(8.98930)
MOVL C00092 V=30.0 PL=1
'ExtruderHandler(9.14602)
MOVL C00093 V=30.0 PL=1
'ExtruderHandler(9.30275)
MOVL C00094 V=30.0 PL=1
'ExtruderHandler(9.45947)
MOVL C00095 V=30.0 PL=1
'ExtruderHandler(9.61619)
MOVL C00096 V=30.0 PL=1
'ExtruderHandler(9.77292)
MOVL C00097 V=30.0 PL=1
'ExtruderHandler(9.92964)
MOVL C00098 V=30.0 PL=1
'ExtruderHandler(10.08636)
MOVL C00099 V=30.0 PL=1
'ExtruderHandler(10.15917)
MOVL C00100 V=30.0 PL=1
MOVL C00101 V=130.0 PL=1
'ExtruderHandler(10.23373)
MOVL C00102 V=30.0 PL=1
'ExtruderHandler(10.39542)
MOVL C00103 V=30.0 PL=1
'ExtruderHandler(10.55712)
MOVL C00104 V=30.0 PL=1
'ExtruderHandler(10.71881)
MOVL C00105 V=30.0 PL=1
'ExtruderHandler(10.88050)
MOVL C00106 V=30.0 PL=1
'ExtruderHandler(11.04220)
MOVL C00107 V=30.0 PL=1
'ExtruderHandler(11.20389)
MOVL C00108 V=30.0 PL=1
'ExtruderHandler(11.36558)
MOVL C00109 V=30.0 PL=1
'ExtruderHandler(11.52727)
MOVL C00110 V=30.0 PL=1
'ExtruderHandler(11.68897)
MOVL C00111 V=30.0 PL=1
'ExtruderHandler(11.85066)
MOVL C00112 V=30.0 PL=1
'ExtruderHandler(12.01235)
MOVL C00113 V=30.0 PL=1
'ExtruderHandler(12.17405)
MOVL C00114 V=30.0 PL=1
'ExtruderHandler(12.33574)
MOVL C00115 V=30.0 PL=1
'ExtruderHandler(12.49743)
MOVL C00116 V=30.0 PL=1
'ExtruderHandler(12.65913)
MOVL C00117 V=30.0 PL=1
'ExtruderHandler(12.82082)
MOVL C00118 V=30.0 PL=1
'ExtruderHandler(12.98251)
MOVL C00119 V=30.0 PL=1
'ExtruderHandler(13.05781)
MOVL C00120 V=30.0 PL=1
MOVL C00121 V=130.0 PL=1
'ExtruderHandler(11.05781)
'ExtruderHandler(0.00000)
MOVL C00122 V=130.0 PL=1
'ExtruderHandler(2.00000)
'ExtruderHandler(2.01570)
MOVL C00123 V=30.0 PL=1
'ExtruderHandler(2.07155)
MOVL C00124 V=30.0 PL=1
'ExtruderHandler(2.28846)
MOVL C00125 V=30.0 PL=1
'ExtruderHandler(2.32266)
MOVL C00126 V=30.0 PL=1
'ExtruderHandler(2.62452)
MOVL C00127 V=30.0 PL=1
'ExtruderHandler(2.65643)
MOVL C00128 V=30.0 PL=1
'ExtruderHandler(2.66723)
MOVL C00129 V=30.0 PL=1
'ExtruderHandler(3.03977)
MOVL C00130 V=30.0 PL=1
'ExtruderHandler(3.07397)
MOVL C00131 V=30.0 PL=1
'ExtruderHandler(3.49815)
MOVL C00132 V=30.0 PL=1
'ExtruderHandler(3.52335)
MOVL C00133 V=30.0 PL=1
'ExtruderHandler(3.99917)
MOVL C00134 V=30.0 PL=1
'ExtruderHandler(4.00139)
MOVL C00135 V=30.0 PL=1
'ExtruderHandler(4.02051)
MOVL C00136 V=30.0 PL=1
'ExtruderHandler(4.53251)
MOVL C00137 V=30.0 PL=1
'ExtruderHandler(4.55771)
MOVL C00138 V=30.0 PL=1
'ExtruderHandler(5.10481)
MOVL C00139 V=30.0 PL=1
'ExtruderHandler(5.12525)
MOVL C00140 V=30.0 PL=1
'ExtruderHandler(5.70745)
MOVL C00141 V=30.0 PL=1
'ExtruderHandler(5.71427)
MOVL C00142 V=30.0 PL=1
'ExtruderHandler(5.72714)
MOVL C00143 V=30.0 PL=1
'ExtruderHandler(6.33677)
MOVL C00144 V=30.0 PL=1
'ExtruderHandler(6.35721)
MOVL C00145 V=30.0 PL=1
'ExtruderHandler(6.99141)
MOVL C00146 V=30.0 PL=1
'ExtruderHandler(7.00906)
MOVL C00147 V=30.0 PL=1
'ExtruderHandler(7.66784)
MOVL C00148 V=30.0 PL=1
'ExtruderHandler(7.68828)
MOVL C00149 V=30.0 PL=1
'ExtruderHandler(8.37164)
MOVL C00150 V=30.0 PL=1
'ExtruderHandler(8.38928)
MOVL C00151 V=30.0 PL=1
'ExtruderHandler(9.09020)
MOVL C00152 V=30.0 PL=1
'ExtruderHandler(9.10615)
MOVL C00153 V=30.0 PL=1
'ExtruderHandler(9.82393)
MOVL C00154 V=30.0 PL=1
'ExtruderHandler(9.84158)
MOVL C00155 V=30.0 PL=1
'ExtruderHandler(10.57622)
MOVL C00156 V=30.0 PL=1
'ExtruderHandler(10.59217)
MOVL C00157 V=30.0 PL=1
'ExtruderHandler(11.34368)
MOVL C00158 V=30.0 PL=1
'ExtruderHandler(11.35090)
MOVL C00159 V=30.0 PL=1
'ExtruderHandler(11.35975)
MOVL C00160 V=30.0 PL=1
'ExtruderHandler(12.12442)
MOVL C00161 V=30.0 PL=1
'ExtruderHandler(12.14037)
MOVL C00162 V=30.0 PL=1
'ExtruderHandler(12.91567)
MOVL C00163 V=30.0 PL=1
'ExtruderHandler(12.93063)
MOVL C00164 V=30.0 PL=1
'ExtruderHandler(13.71654)
MOVL C00165 V=30.0 PL=1
'ExtruderHandler(13.73249)
MOVL C00166 V=30.0 PL=1
'ExtruderHandler(14.52901)
MOVL C00167 V=30.0 PL=1
'ExtruderHandler(14.54398)
MOVL C00168 V=30.0 PL=1
'ExtruderHandler(15.35112)
MOVL C00169 V=30.0 PL=1
'ExtruderHandler(15.35264)
MOVL C00170 V=30.0 PL=1
'ExtruderHandler(15.36576)
MOVL C00171 V=30.0 PL=1
'ExtruderHandler(16.17856)
MOVL C00172 V=30.0 PL=1
'ExtruderHandler(16.19353)
MOVL C00173 V=30.0 PL=1
'ExtruderHandler(17.01146)
MOVL C00174 V=30.0 PL=1
'ExtruderHandler(17.02597)
MOVL C00175 V=30.0 PL=1
'ExtruderHandler(17.84905)
MOVL C00176 V=30.0 PL=1
'ExtruderHandler(17.86401)
MOVL C00177 V=30.0 PL=1
'ExtruderHandler(18.69223)
MOVL C00178 V=30.0 PL=1
'ExtruderHandler(18.70674)
MOVL C00179 V=30.0 PL=1
'ExtruderHandler(19.54009)
MOVL C00180 V=30.0 PL=1
'ExtruderHandler(19.55459)
MOVL C00181 V=30.0 PL=1
'ExtruderHandler(20.38798)
MOVL C00182 V=30.0 PL=1
'ExtruderHandler(20.40249)
MOVL C00183 V=30.0 PL=1
'ExtruderHandler(21.23587)
MOVL C00184 V=30.0 PL=1
'ExtruderHandler(21.25038)
MOVL C00185 V=30.0 PL=1
'ExtruderHandler(22.08377)
MOVL C00186 V=30.0 PL=1
'ExtruderHandler(22.09828)
MOVL C00187 V=30.0 PL=1
'ExtruderHandler(22.93166)
MOVL C00188 V=30.0 PL=1
'ExtruderHandler(22.94617)
MOVL C00189 V=30.0 PL=1
'ExtruderHandler(23.77952)
MOVL C00190 V=30.0 PL=1
'ExtruderHandler(23.79449)
MOVL C00191 V=30.0 PL=1
'ExtruderHandler(24.62270)
MOVL C00192 V=30.0 PL=1
'ExtruderHandler(24.63721)
MOVL C00193 V=30.0 PL=1
'ExtruderHandler(25.46028)
MOVL C00194 V=30.0 PL=1
'ExtruderHandler(25.47525)
MOVL C00195 V=30.0 PL=1
'ExtruderHandler(26.29319)
MOVL C00196 V=30.0 PL=1
'ExtruderHandler(26.30770)
MOVL C00197 V=30.0 PL=1
'ExtruderHandler(27.12049)
MOVL C00198 V=30.0 PL=1
'ExtruderHandler(27.13546)
MOVL C00199 V=30.0 PL=1
'ExtruderHandler(27.94260)
MOVL C00200 V=30.0 PL=1
'ExtruderHandler(27.95855)
MOVL C00201 V=30.0 PL=1
'ExtruderHandler(28.75507)
MOVL C00202 V=30.0 PL=1
'ExtruderHandler(28.77003)
MOVL C00203 V=30.0 PL=1
'ExtruderHandler(29.55594)
MOVL C00204 V=30.0 PL=1
'ExtruderHandler(29.57189)
MOVL C00205 V=30.0 PL=1
'ExtruderHandler(30.34718)
MOVL C00206 V=30.0 PL=1
'ExtruderHandler(30.36215)
MOVL C00207 V=30.0 PL=1
'ExtruderHandler(31.12683)
MOVL C00208 V=30.0 PL=1
'ExtruderHandler(31.14278)
MOVL C00209 V=30.0 PL=1
'ExtruderHandler(31.89428)
MOVL C00210 V=30.0 PL=1
'ExtruderHandler(31.91193)
MOVL C00211 V=30.0 PL=1
'ExtruderHandler(32.64658)
MOVL C00212 V=30.0 PL=1
'ExtruderHandler(32.66253)
MOVL C00213 V=30.0 PL=1
'ExtruderHandler(33.38031)
MOVL C00214 V=30.0 PL=1
'ExtruderHandler(33.39795)
MOVL C00215 V=30.0 PL=1
'ExtruderHandler(34.09887)
MOVL C00216 V=30.0 PL=1
'ExtruderHandler(34.11338)
MOVL C00217 V=30.0 PL=1
'ExtruderHandler(34.11523)
MOVL C00218 V=30.0 PL=1
'ExtruderHandler(34.79858)
MOVL C00219 V=30.0 PL=1
'ExtruderHandler(34.81623)
MOVL C00220 V=30.0 PL=1
'ExtruderHandler(35.47501)
MOVL C00221 V=30.0 PL=1
'ExtruderHandler(35.49545)
MOVL C00222 V=30.0 PL=1
'ExtruderHandler(36.12965)
MOVL C00223 V=30.0 PL=1
'ExtruderHandler(36.14730)
MOVL C00224 V=30.0 PL=1
'ExtruderHandler(36.75692)
MOVL C00225 V=30.0 PL=1
'ExtruderHandler(36.77737)
MOVL C00226 V=30.0 PL=1
'ExtruderHandler(37.35956)
MOVL C00227 V=30.0 PL=1
'ExtruderHandler(37.38477)
MOVL C00228 V=30.0 PL=1
'ExtruderHandler(37.93186)
MOVL C00229 V=30.0 PL=1
'ExtruderHandler(37.95231)
MOVL C00230 V=30.0 PL=1
'ExtruderHandler(38.46430)
MOVL C00231 V=30.0 PL=1
'ExtruderHandler(38.48951)
MOVL C00232 V=30.0 PL=1
'ExtruderHandler(38.96533)
MOVL C00233 V=30.0 PL=1
'ExtruderHandler(38.99953)
MOVL C00234 V=30.0 PL=1
'ExtruderHandler(39.42371)
MOVL C00235 V=30.0 PL=1
'ExtruderHandler(39.44891)
MOVL C00236 V=30.0 PL=1
'ExtruderHandler(39.82144)
MOVL C00237 V=30.0 PL=1
'ExtruderHandler(39.85565)
MOVL C00238 V=30.0 PL=1
'ExtruderHandler(40.15750)
MOVL C00239 V=30.0 PL=1
'ExtruderHandler(40.21335)
MOVL C00240 V=30.0 PL=1
'ExtruderHandler(40.43025)
MOVL C00241 V=30.0 PL=1
'ExtruderHandler(40.43484)
MOVL C00242 V=30.0 PL=1
'ExtruderHandler(40.57845)
MOVL C00243 V=30.0 PL=1
'ExtruderHandler(40.59417)
MOVL C00244 V=30.0 PL=1
'MCodeHandler(104)
MOVL C00245 V=130.0 PL=1
MOVL C00246 V=130.0 PL=1
'ExtruderHandler(40.79179)
MOVL C00247 V=60.0 PL=1
'ExtruderHandler(41.26492)
MOVL C00248 V=60.0 PL=1
'ExtruderHandler(41.73805)
MOVL C00249 V=60.0 PL=1
'ExtruderHandler(42.21118)
MOVL C00250 V=60.0 PL=1
'ExtruderHandler(42.68431)
MOVL C00251 V=60.0 PL=1
'ExtruderHandler(43.15744)
MOVL C00252 V=60.0 PL=1
'ExtruderHandler(43.63057)
MOVL C00253 V=60.0 PL=1
'ExtruderHandler(44.10370)
MOVL C00254 V=60.0 PL=1
'ExtruderHandler(44.57683)
MOVL C00255 V=60.0 PL=1
'ExtruderHandler(45.04996)
MOVL C00256 V=60.0 PL=1
'ExtruderHandler(45.52309)
MOVL C00257 V=60.0 PL=1
'ExtruderHandler(45.99622)
MOVL C00258 V=60.0 PL=1
'ExtruderHandler(46.46935)
MOVL C00259 V=60.0 PL=1
'ExtruderHandler(46.94248)
MOVL C00260 V=60.0 PL=1
'ExtruderHandler(47.41561)
MOVL C00261 V=60.0 PL=1
'ExtruderHandler(47.88874)
MOVL C00262 V=60.0 PL=1
'ExtruderHandler(48.36187)
MOVL C00263 V=60.0 PL=1
'ExtruderHandler(48.83500)
MOVL C00264 V=60.0 PL=1
'ExtruderHandler(49.03715)
MOVL C00265 V=60.0 PL=1
MOVL C00266 V=130.0 PL=1
'ExtruderHandler(49.35402)
MOVL C00267 V=60.0 PL=1
'ExtruderHandler(50.06565)
MOVL C00268 V=60.0 PL=1
'ExtruderHandler(50.77728)
MOVL C00269 V=60.0 PL=1
'ExtruderHandler(51.48892)
MOVL C00270 V=60.0 PL=1
'ExtruderHandler(52.20055)
MOVL C00271 V=60.0 PL=1
'ExtruderHandler(52.91219)
MOVL C00272 V=60.0 PL=1
'ExtruderHandler(53.62382)
MOVL C00273 V=60.0 PL=1
'ExtruderHandler(54.33545)
MOVL C00274 V=60.0 PL=1
'ExtruderHandler(55.04709)
MOVL C00275 V=60.0 PL=1
'ExtruderHandler(55.75872)
MOVL C00276 V=60.0 PL=1
'ExtruderHandler(56.47035)
MOVL C00277 V=60.0 PL=1
'ExtruderHandler(57.18199)
MOVL C00278 V=60.0 PL=1
'ExtruderHandler(57.89362)
MOVL C00279 V=60.0 PL=1
'ExtruderHandler(58.60526)
MOVL C00280 V=60.0 PL=1
'ExtruderHandler(59.31689)
MOVL C00281 V=60.0 PL=1
'ExtruderHandler(60.02852)
MOVL C00282 V=60.0 PL=1
'ExtruderHandler(60.74016)
MOVL C00283 V=60.0 PL=1
'ExtruderHandler(61.45179)
MOVL C00284 V=60.0 PL=1
'ExtruderHandler(61.77320)
MOVL C00285 V=60.0 PL=1
MOVL C00286 V=130.0 PL=1
'ExtruderHandler(62.10457)
MOVL C00287 V=30.0 PL=1
'ExtruderHandler(62.82832)
MOVL C00288 V=30.0 PL=1
'ExtruderHandler(63.55207)
MOVL C00289 V=30.0 PL=1
'ExtruderHandler(64.27582)
MOVL C00290 V=30.0 PL=1
'ExtruderHandler(64.99957)
MOVL C00291 V=30.0 PL=1
'ExtruderHandler(65.72332)
MOVL C00292 V=30.0 PL=1
'ExtruderHandler(66.44707)
MOVL C00293 V=30.0 PL=1
'ExtruderHandler(67.17082)
MOVL C00294 V=30.0 PL=1
'ExtruderHandler(67.89457)
MOVL C00295 V=30.0 PL=1
'ExtruderHandler(68.61832)
MOVL C00296 V=30.0 PL=1
'ExtruderHandler(69.34207)
MOVL C00297 V=30.0 PL=1
'ExtruderHandler(70.06582)
MOVL C00298 V=30.0 PL=1
'ExtruderHandler(70.78957)
MOVL C00299 V=30.0 PL=1
'ExtruderHandler(71.51332)
MOVL C00300 V=30.0 PL=1
'ExtruderHandler(72.23708)
MOVL C00301 V=30.0 PL=1
'ExtruderHandler(72.96083)
MOVL C00302 V=30.0 PL=1
'ExtruderHandler(73.68458)
MOVL C00303 V=30.0 PL=1
'ExtruderHandler(74.40833)
MOVL C00304 V=30.0 PL=1
'ExtruderHandler(74.74326)
MOVL C00305 V=30.0 PL=1
MOVL C00306 V=130.0 PL=1
MOVL C00307 V=130.0 PL=1
'ExtruderHandler(77.20486)
MOVL C00308 V=20.0 PL=1
MOVL C00309 V=130.0 PL=1
'ExtruderHandler(78.09759)
MOVL C00310 V=20.0 PL=1
MOVL C00311 V=130.0 PL=1
MOVL C00312 V=130.0 PL=1
'ExtruderHandler(78.29520)
MOVL C00313 V=60.0 PL=1
'ExtruderHandler(78.76833)
MOVL C00314 V=60.0 PL=1
'ExtruderHandler(79.24146)
MOVL C00315 V=60.0 PL=1
'ExtruderHandler(79.71459)
MOVL C00316 V=60.0 PL=1
'ExtruderHandler(80.18772)
MOVL C00317 V=60.0 PL=1
'ExtruderHandler(80.66085)
MOVL C00318 V=60.0 PL=1
'ExtruderHandler(81.13398)
MOVL C00319 V=60.0 PL=1
'ExtruderHandler(81.60711)
MOVL C00320 V=60.0 PL=1
'ExtruderHandler(82.08024)
MOVL C00321 V=60.0 PL=1
'ExtruderHandler(82.55337)
MOVL C00322 V=60.0 PL=1
'ExtruderHandler(83.02650)
MOVL C00323 V=60.0 PL=1
'ExtruderHandler(83.49963)
MOVL C00324 V=60.0 PL=1
'ExtruderHandler(83.97276)
MOVL C00325 V=60.0 PL=1
'ExtruderHandler(84.44589)
MOVL C00326 V=60.0 PL=1
'ExtruderHandler(84.91902)
MOVL C00327 V=60.0 PL=1
'ExtruderHandler(85.39215)
MOVL C00328 V=60.0 PL=1
'ExtruderHandler(85.86528)
MOVL C00329 V=60.0 PL=1
'ExtruderHandler(86.33841)
MOVL C00330 V=60.0 PL=1
'ExtruderHandler(86.54057)
MOVL C00331 V=60.0 PL=1
MOVL C00332 V=130.0 PL=1
'ExtruderHandler(86.85743)
MOVL C00333 V=60.0 PL=1
'ExtruderHandler(87.56907)
MOVL C00334 V=60.0 PL=1
'ExtruderHandler(88.28070)
MOVL C00335 V=60.0 PL=1
'ExtruderHandler(88.99233)
MOVL C00336 V=60.0 PL=1
'ExtruderHandler(89.70397)
MOVL C00337 V=60.0 PL=1
'ExtruderHandler(90.41560)
MOVL C00338 V=60.0 PL=1
'ExtruderHandler(91.12724)
MOVL C00339 V=60.0 PL=1
'ExtruderHandler(91.83887)
MOVL C00340 V=60.0 PL=1
'ExtruderHandler(92.55050)
MOVL C00341 V=60.0 PL=1
'ExtruderHandler(93.26214)
MOVL C00342 V=60.0 PL=1
'ExtruderHandler(93.97377)
MOVL C00343 V=60.0 PL=1
'ExtruderHandler(94.68540)
MOVL C00344 V=60.0 PL=1
'ExtruderHandler(95.39704)
MOVL C00345 V=60.0 PL=1
'ExtruderHandler(96.10867)
MOVL C00346 V=60.0 PL=1
'ExtruderHandler(96.82031)
MOVL C00347 V=60.0 PL=1
'ExtruderHandler(97.53194)
MOVL C00348 V=60.0 PL=1
'ExtruderHandler(98.24357)
MOVL C00349 V=60.0 PL=1
'ExtruderHandler(98.95521)
MOVL C00350 V=60.0 PL=1
'ExtruderHandler(99.27662)
MOVL C00351 V=60.0 PL=1
MOVL C00352 V=130.0 PL=1
'ExtruderHandler(99.60799)
MOVL C00353 V=30.0 PL=1
'ExtruderHandler(100.33174)
MOVL C00354 V=30.0 PL=1
'ExtruderHandler(101.05549)
MOVL C00355 V=30.0 PL=1
'ExtruderHandler(101.77924)
MOVL C00356 V=30.0 PL=1
'ExtruderHandler(102.50299)
MOVL C00357 V=30.0 PL=1
'ExtruderHandler(103.22674)
MOVL C00358 V=30.0 PL=1
'ExtruderHandler(103.95049)
MOVL C00359 V=30.0 PL=1
'ExtruderHandler(104.67424)
MOVL C00360 V=30.0 PL=1
'ExtruderHandler(105.39799)
MOVL C00361 V=30.0 PL=1
'ExtruderHandler(106.12174)
MOVL C00362 V=30.0 PL=1
'ExtruderHandler(106.84549)
MOVL C00363 V=30.0 PL=1
'ExtruderHandler(107.56924)
MOVL C00364 V=30.0 PL=1
'ExtruderHandler(108.29299)
MOVL C00365 V=30.0 PL=1
'ExtruderHandler(109.01674)
MOVL C00366 V=30.0 PL=1
'ExtruderHandler(109.74049)
MOVL C00367 V=30.0 PL=1
'ExtruderHandler(110.46424)
MOVL C00368 V=30.0 PL=1
'ExtruderHandler(111.18799)
MOVL C00369 V=30.0 PL=1
'ExtruderHandler(111.91174)
MOVL C00370 V=30.0 PL=1
'ExtruderHandler(112.24667)
MOVL C00371 V=30.0 PL=1
MOVL C00372 V=130.0 PL=1
MOVL C00373 V=130.0 PL=1
'ExtruderHandler(112.42380)
MOVL C00374 V=20.0 PL=1
'ExtruderHandler(112.70535)
MOVL C00375 V=20.0 PL=1
'ExtruderHandler(112.98690)
MOVL C00376 V=20.0 PL=1
'ExtruderHandler(113.26845)
MOVL C00377 V=20.0 PL=1
'ExtruderHandler(113.55001)
MOVL C00378 V=20.0 PL=1
'ExtruderHandler(113.83156)
MOVL C00379 V=20.0 PL=1
'ExtruderHandler(114.11311)
MOVL C00380 V=20.0 PL=1
'ExtruderHandler(114.39466)
MOVL C00381 V=20.0 PL=1
'ExtruderHandler(114.43310)
MOVL C00382 V=20.0 PL=1
'ExtruderHandler(116.89284)
MOVL C00383 V=20.0 PL=1
'ExtruderHandler(116.99727)
MOVL C00384 V=20.0 PL=1
'ExtruderHandler(117.27883)
MOVL C00385 V=20.0 PL=1
'ExtruderHandler(117.56038)
MOVL C00386 V=20.0 PL=1
'ExtruderHandler(117.84193)
MOVL C00387 V=20.0 PL=1
'ExtruderHandler(118.12348)
MOVL C00388 V=20.0 PL=1
'ExtruderHandler(118.34475)
MOVL C00389 V=20.0 PL=1
'ExtruderHandler(119.23763)
MOVL C00390 V=20.0 PL=1
'MCodeHandler(106)
MOVL C00391 V=130.0 PL=1
MOVL C00392 V=130.0 PL=1
'ExtruderHandler(119.43524)
MOVL C00393 V=60.0 PL=1
'ExtruderHandler(119.90837)
MOVL C00394 V=60.0 PL=1
'ExtruderHandler(120.38150)
MOVL C00395 V=60.0 PL=1
'ExtruderHandler(120.85463)
MOVL C00396 V=60.0 PL=1
'ExtruderHandler(121.32776)
MOVL C00397 V=60.0 PL=1
'ExtruderHandler(121.80089)
MOVL C00398 V=60.0 PL=1
'ExtruderHandler(122.27402)
MOVL C00399 V=60.0 PL=1
'ExtruderHandler(122.74715)
MOVL C00400 V=60.0 PL=1
'ExtruderHandler(123.22028)
MOVL C00401 V=60.0 PL=1
'ExtruderHandler(123.69341)
MOVL C00402 V=60.0 PL=1
'ExtruderHandler(124.16654)
MOVL C00403 V=60.0 PL=1
'ExtruderHandler(124.63967)
MOVL C00404 V=60.0 PL=1
'ExtruderHandler(125.11280)
MOVL C00405 V=60.0 PL=1
'ExtruderHandler(125.58593)
MOVL C00406 V=60.0 PL=1
'ExtruderHandler(126.05906)
MOVL C00407 V=60.0 PL=1
'ExtruderHandler(126.53219)
MOVL C00408 V=60.0 PL=1
'ExtruderHandler(127.00532)
MOVL C00409 V=60.0 PL=1
'ExtruderHandler(127.47845)
MOVL C00410 V=60.0 PL=1
'ExtruderHandler(127.68061)
MOVL C00411 V=60.0 PL=1
MOVL C00412 V=130.0 PL=1
'ExtruderHandler(127.99747)
MOVL C00413 V=60.0 PL=1
'ExtruderHandler(128.70911)
MOVL C00414 V=60.0 PL=1
'ExtruderHandler(129.42074)
MOVL C00415 V=60.0 PL=1
'ExtruderHandler(130.13237)
MOVL C00416 V=60.0 PL=1
'ExtruderHandler(130.84401)
MOVL C00417 V=60.0 PL=1
'ExtruderHandler(131.55564)
MOVL C00418 V=60.0 PL=1
'ExtruderHandler(132.26728)
MOVL C00419 V=60.0 PL=1
'ExtruderHandler(132.97891)
MOVL C00420 V=60.0 PL=1
'ExtruderHandler(133.69054)
MOVL C00421 V=60.0 PL=1
'ExtruderHandler(134.40218)
MOVL C00422 V=60.0 PL=1
'ExtruderHandler(135.11381)
MOVL C00423 V=60.0 PL=1
'ExtruderHandler(135.82544)
MOVL C00424 V=60.0 PL=1
'ExtruderHandler(136.53708)
MOVL C00425 V=60.0 PL=1
'ExtruderHandler(137.24871)
MOVL C00426 V=60.0 PL=1
'ExtruderHandler(137.96035)
MOVL C00427 V=60.0 PL=1
'ExtruderHandler(138.67198)
MOVL C00428 V=60.0 PL=1
'ExtruderHandler(139.38361)
MOVL C00429 V=60.0 PL=1
'ExtruderHandler(140.09525)
MOVL C00430 V=60.0 PL=1
'ExtruderHandler(140.41666)
MOVL C00431 V=60.0 PL=1
MOVL C00432 V=130.0 PL=1
'ExtruderHandler(140.74803)
MOVL C00433 V=30.0 PL=1
'ExtruderHandler(141.47178)
MOVL C00434 V=30.0 PL=1
'ExtruderHandler(142.19553)
MOVL C00435 V=30.0 PL=1
'ExtruderHandler(142.91928)
MOVL C00436 V=30.0 PL=1
'ExtruderHandler(143.64303)
MOVL C00437 V=30.0 PL=1
'ExtruderHandler(144.36678)
MOVL C00438 V=30.0 PL=1
'ExtruderHandler(145.09053)
MOVL C00439 V=30.0 PL=1
'ExtruderHandler(145.81428)
MOVL C00440 V=30.0 PL=1
'ExtruderHandler(146.53803)
MOVL C00441 V=30.0 PL=1
'ExtruderHandler(147.26178)
MOVL C00442 V=30.0 PL=1
'ExtruderHandler(147.98553)
MOVL C00443 V=30.0 PL=1
'ExtruderHandler(148.70928)
MOVL C00444 V=30.0 PL=1
'ExtruderHandler(149.43303)
MOVL C00445 V=30.0 PL=1
'ExtruderHandler(150.15678)
MOVL C00446 V=30.0 PL=1
'ExtruderHandler(150.88053)
MOVL C00447 V=30.0 PL=1
'ExtruderHandler(151.60428)
MOVL C00448 V=30.0 PL=1
'ExtruderHandler(152.32803)
MOVL C00449 V=30.0 PL=1
'ExtruderHandler(153.05178)
MOVL C00450 V=30.0 PL=1
'ExtruderHandler(153.38671)
MOVL C00451 V=30.0 PL=1
MOVL C00452 V=130.0 PL=1
MOVL C00453 V=130.0 PL=1
'ExtruderHandler(155.84832)
MOVL C00454 V=20.0 PL=1
MOVL C00455 V=130.0 PL=1
'ExtruderHandler(156.74105)
MOVL C00456 V=20.0 PL=1
'MCodeHandler(106)
MOVL C00457 V=130.0 PL=1
'ExtruderHandler(154.74105)
'ExtruderHandler(0.00000)
MOVL C00458 V=130.0 PL=1
'ExtruderHandler(2.00000)
'ExtruderHandler(2.19761)
MOVL C00459 V=60.0 PL=1
'ExtruderHandler(2.67074)
MOVL C00460 V=60.0 PL=1
'ExtruderHandler(3.14387)
MOVL C00461 V=60.0 PL=1
'ExtruderHandler(3.61700)
MOVL C00462 V=60.0 PL=1
'ExtruderHandler(4.09013)
MOVL C00463 V=60.0 PL=1
'ExtruderHandler(4.56326)
MOVL C00464 V=60.0 PL=1
'ExtruderHandler(5.03639)
MOVL C00465 V=60.0 PL=1
'ExtruderHandler(5.50952)
MOVL C00466 V=60.0 PL=1
'ExtruderHandler(5.98265)
MOVL C00467 V=60.0 PL=1
'ExtruderHandler(6.45578)
MOVL C00468 V=60.0 PL=1
'ExtruderHandler(6.92891)
MOVL C00469 V=60.0 PL=1
'ExtruderHandler(7.40204)
MOVL C00470 V=60.0 PL=1
'ExtruderHandler(7.87517)
MOVL C00471 V=60.0 PL=1
'ExtruderHandler(8.34830)
MOVL C00472 V=60.0 PL=1
'ExtruderHandler(8.82143)
MOVL C00473 V=60.0 PL=1
'ExtruderHandler(9.29456)
MOVL C00474 V=60.0 PL=1
'ExtruderHandler(9.76769)
MOVL C00475 V=60.0 PL=1
'ExtruderHandler(10.24082)
MOVL C00476 V=60.0 PL=1
'ExtruderHandler(10.44298)
MOVL C00477 V=60.0 PL=1
'ExtruderHandler(8.44298)
'ExtruderHandler(0.00000)
MOVL C00478 V=130.0 PL=1
'ExtruderHandler(2.00000)
'ExtruderHandler(2.31686)
MOVL C00479 V=60.0 PL=1
'ExtruderHandler(3.02850)
MOVL C00480 V=60.0 PL=1
'ExtruderHandler(3.74013)
MOVL C00481 V=60.0 PL=1
'ExtruderHandler(4.45176)
MOVL C00482 V=60.0 PL=1
'ExtruderHandler(5.16340)
MOVL C00483 V=60.0 PL=1
'ExtruderHandler(5.87503)
MOVL C00484 V=60.0 PL=1
'ExtruderHandler(6.58667)
MOVL C00485 V=60.0 PL=1
'ExtruderHandler(7.29830)
MOVL C00486 V=60.0 PL=1
'ExtruderHandler(8.00993)
MOVL C00487 V=60.0 PL=1
'ExtruderHandler(8.72157)
MOVL C00488 V=60.0 PL=1
'ExtruderHandler(9.43320)
MOVL C00489 V=60.0 PL=1
'ExtruderHandler(10.14483)
MOVL C00490 V=60.0 PL=1
'ExtruderHandler(10.85647)
MOVL C00491 V=60.0 PL=1
'ExtruderHandler(11.56810)
MOVL C00492 V=60.0 PL=1
'ExtruderHandler(12.27974)
MOVL C00493 V=60.0 PL=1
'ExtruderHandler(12.99137)
MOVL C00494 V=60.0 PL=1
'ExtruderHandler(13.70300)
MOVL C00495 V=60.0 PL=1
'ExtruderHandler(14.41464)
MOVL C00496 V=60.0 PL=1
'ExtruderHandler(14.73605)
MOVL C00497 V=60.0 PL=1
'ExtruderHandler(12.73605)
'ExtruderHandler(0.00000)
MOVL C00498 V=130.0 PL=1
'ExtruderHandler(2.00000)
'ExtruderHandler(2.33137)
MOVL C00499 V=30.0 PL=1
'ExtruderHandler(3.05512)
MOVL C00500 V=30.0 PL=1
'ExtruderHandler(3.77887)
MOVL C00501 V=30.0 PL=1
'ExtruderHandler(4.50262)
MOVL C00502 V=30.0 PL=1
'ExtruderHandler(5.22637)
MOVL C00503 V=30.0 PL=1
'ExtruderHandler(5.95012)
MOVL C00504 V=30.0 PL=1
'ExtruderHandler(6.67387)
MOVL C00505 V=30.0 PL=1
'ExtruderHandler(7.39762)
MOVL C00506 V=30.0 PL=1
'ExtruderHandler(8.12137)
MOVL C00507 V=30.0 PL=1
'ExtruderHandler(8.84512)
MOVL C00508 V=30.0 PL=1
'ExtruderHandler(9.56888)
MOVL C00509 V=30.0 PL=1
'ExtruderHandler(10.29263)
MOVL C00510 V=30.0 PL=1
'ExtruderHandler(11.01638)
MOVL C00511 V=30.0 PL=1
'ExtruderHandler(11.74013)
MOVL C00512 V=30.0 PL=1
'ExtruderHandler(12.46388)
MOVL C00513 V=30.0 PL=1
'ExtruderHandler(13.18763)
MOVL C00514 V=30.0 PL=1
'ExtruderHandler(13.91138)
MOVL C00515 V=30.0 PL=1
'ExtruderHandler(14.63513)
MOVL C00516 V=30.0 PL=1
'ExtruderHandler(14.97006)
MOVL C00517 V=30.0 PL=1
MOVL C00518 V=130.0 PL=1
'ExtruderHandler(12.97006)
'ExtruderHandler(0.00000)
MOVL C00519 V=130.0 PL=1
'ExtruderHandler(2.00000)
'ExtruderHandler(2.18255)
MOVL C00520 V=15.0 PL=1
'ExtruderHandler(2.46410)
MOVL C00521 V=15.0 PL=1
'ExtruderHandler(2.74565)
MOVL C00522 V=15.0 PL=1
'ExtruderHandler(3.02721)
MOVL C00523 V=15.0 PL=1
'ExtruderHandler(3.30876)
MOVL C00524 V=15.0 PL=1
'ExtruderHandler(3.59031)
MOVL C00525 V=15.0 PL=1
'ExtruderHandler(3.87186)
MOVL C00526 V=15.0 PL=1
'ExtruderHandler(4.15342)
MOVL C00527 V=15.0 PL=1
'ExtruderHandler(4.19712)
MOVL C00528 V=15.0 PL=1
'ExtruderHandler(6.65872)
MOVL C00529 V=15.0 PL=1
'ExtruderHandler(6.75773)
MOVL C00530 V=15.0 PL=1
'ExtruderHandler(7.03928)
MOVL C00531 V=15.0 PL=1
'ExtruderHandler(7.32083)
MOVL C00532 V=15.0 PL=1
'ExtruderHandler(7.60238)
MOVL C00533 V=15.0 PL=1
'ExtruderHandler(7.88394)
MOVL C00534 V=15.0 PL=1
'ExtruderHandler(8.16535)
MOVL C00535 V=15.0 PL=1
'ExtruderHandler(9.05826)
MOVL C00536 V=15.0 PL=1
'ExtruderHandler(7.05826)
MOVL C00537 V=40.0 PL=1
'ExtruderHandler(0.00000)
'MCodeHandler(107)
'MCodeHandler(104)
'MCodeHandler(84)
'MCodeHandler(140)
END
